// TIA Portal V17 export
// export: Created 2024-06-16T17:47:27.9988929Z, ExportSetting WithDefaults, DisplayName Totally Integrated Automation Portal, DisplayVersion V17, DisplayName TIA Portal Openness, DisplayVersion V17, DisplayName TIA Portal Version Control Interface, DisplayVersion V17, DisplayName STEP 7 Professional, DisplayVersion V17, DisplayName STEP 7 Safety, DisplayVersion V17, DisplayName WinCC Professional, DisplayVersion V17
DATA_BLOCK "St2_In"   // DB205
{ S7_Optimized_Access := 'TRUE' }
VERSION : 0.1
// stored: AutoNumber false, DBAccessibleFromOPCUA true, DBAccessibleFromWebserver true, IsOnlyStoredInLoadMemory false, IsRetainMemResEnabled false, IsWriteProtectedInAS false, MemoryReserve 100
   VAR
      Cpt_V1 : Bool;   // Présence barquette en début de Vision : V1
      Cpt_V2 : Bool;   // Détection butée à came : V2
      Cpt_V3 : Bool;   // Détection butée pivot : V3
   END_VAR
BEGIN
END_DATA_BLOCK
